FUNCTION_BLOCK Zebra
VAR_INPUT
END_VAR
VAR_OUTPUT
END_VAR
VAR
END_VAR

END_FUNCTION_BLOCK

(* stored: Version 1.1.0.1, ProductVersion 3.1.4024.12
   POU Zebra: Id {b531e07b-7a9a-45c7-85a0-6696bc7d2a01}, SpecialFunc None *)
